LIN {X 0,Y 78.039,Z 374.236,A -85,B 0,C 180,E1 -30962.276,E2 -30962.276} C_VEL
LIN {X 0,Y 75.097,Z 386.191,A -85,B 0,C 180,E1 -30962.659,E2 -30962.659} C_VEL
LIN {X 0,Y 70.422,Z 399.419,A -85,B 0,C 180,E1 -30963.507,E2 -30963.507} C_VEL
LIN {X 0,Y 64.332,Z 411.877,A -85,B 0,C 180,E1 -30964.416,E2 -30964.416} C_VEL
LIN {X 0,Y 57.436,Z 423.118,A -85,B 0,C 180,E1 -30966.078,E2 -30966.078} C_VEL
LIN {X 0,Y 49.737,Z 433.18,A -85,B 0,C 180,E1 -30968.373,E2 -30968.373} C_VEL
LIN {X 0,Y 41.305,Z 442.293,A -85,B 0,C 180,E1 -30971.87,E2 -30971.87} C_VEL
LIN {X 0,Y 31.483,Z 451.164,A -85,B 0,C 180,E1 -30978.364,E2 -30978.364} C_VEL
LIN {X 0,Y 22.364,Z 458.209,A -85,B 0,C 180,E1 -30990.155,E2 -30990.155} C_VEL
LIN {X 0,Y 16.168,Z 463.002,A -85,B 0,C 180,E1 -31009.254,E2 -31009.254} C_VEL
LIN {X 0,Y 12.989,Z 467.557,A -85,B 0,C 180,E1 -31049.952,E2 -31049.952} C_VEL
LIN {X 0,Y 14.487,Z 469.9,A -85,B 0,C 180,E1 -31078.972,E2 -31078.972} C_VEL
LIN {X 0,Y 18.537,Z 471.807,A -85,B 0,C 180,E1 -31099.259,E2 -31099.259} C_VEL
LIN {X 0,Y 30.055,Z 474.427,A -85,B 0,C 180,E1 -31119.226,E2 -31119.226} C_VEL
LIN {X 0,Y 43.189,Z 475.464,A -85,B 0,C 180,E1 -31127.447,E2 -31127.447} C_VEL
LIN {X 0,Y 49.96,Z 475.43,A -85,B 0,C 180,E1 -31129.894,E2 -31129.894} C_VEL
LIN {X 0,Y 49.912,Z 475.428,A -85,B 0,C 180,E1 -31130.205,E2 -31130.205} C_VEL
LIN {X 0,Y 42.475,Z 475.388,A -85,B 0,C 180,E1 -31132.983,E2 -31132.983} C_VEL
LIN {X 0,Y 30.984,Z 474.383,A -85,B 0,C 180,E1 -31139.95,E2 -31139.95} C_VEL
LIN {X 0,Y 21.533,Z 472.495,A -85,B 0,C 180,E1 -31151.868,E2 -31151.868} C_VEL
LIN {X 0,Y 13.826,Z 469.451,A -85,B 0,C 180,E1 -31180.388,E2 -31180.388} C_VEL
LIN {X 0,Y 13.127,Z 465.27,A -85,B 0,C 180,E1 -31230.048,E2 -31230.048} C_VEL
LIN {X 0,Y 19.696,Z 459.87,A -85,B 0,C 180,E1 -31262.397,E2 -31262.397} C_VEL
LIN {X 0,Y 28.677,Z 453.089,A -85,B 0,C 180,E1 -31277.359,E2 -31277.359} C_VEL
LIN {X 0,Y 38.527,Z 444.654,A -85,B 0,C 180,E1 -31285.201,E2 -31285.201} C_VEL
LIN {X 0,Y 45.556,Z 437.596,A -85,B 0,C 180,E1 -31288.628,E2 -31288.628} C_VEL
LIN {X 0,Y 49.181,Z 433.304,A -85,B 0,C 180,E1 -31290.888,E2 -31290.888} C_VEL
LIN {X 0,Y 54.376,Z 425.964,A -85,B 0,C 180,E1 -31295.555,E2 -31295.555} C_VEL
LIN {X 0,Y 59.23,Z 418.141,A -85,B 0,C 180,E1 -31299.3,E2 -31299.3} C_VEL
LIN {X 0,Y 62.124,Z 413.092,A -85,B 0,C 180,E1 -31300.314,E2 -31300.314} C_VEL
LIN {X 0,Y 68.321,Z 400.856,A -85,B 0,C 180,E1 -31301.02,E2 -31301.02} C_VEL
LIN {X 0,Y 73.111,Z 388.298,A -85,B 0,C 180,E1 -31301.539,E2 -31301.539} C_VEL
LIN {X 0,Y 76.561,Z 375.283,A -85,B 0,C 180,E1 -31301.809,E2 -31301.809} C_VEL
LIN {X 0,Y 78.852,Z 360.598,A -85,B 0,C 180,E1 -31302.057,E2 -31302.057} C_VEL
LIN {X 0,Y 78.902,Z 359.79,A -85,B 0,C 180,E1 -31302.391,E2 -31302.391} C_VEL
LIN {X 0,Y 78.681,Z 357.8,A -85,B 0,C 180,E1 -31306.83,E2 -31306.83} C_VEL
LIN {X 0,Y 78.732,Z 357.243,A -85,B 0,C 180,E1 -31311.676,E2 -31311.676} C_VEL
LIN {X 0,Y 78.797,Z 357.715,A -85,B 0,C 180,E1 -31313.505,E2 -31313.505} C_VEL
LIN {X 0,Y 78.961,Z 359.812,A -85,B 0,C 180,E1 -31316.818,E2 -31316.818} C_VEL
LIN {X 0,Y 76.701,Z 374.738,A -85,B 0,C 180,E1 -31317.1,E2 -31317.1} C_VEL
LIN {X 0,Y 73.62,Z 386.882,A -85,B 0,C 180,E1 -31317.323,E2 -31317.323} C_VEL
LIN {X 0,Y 69.024,Z 399.468,A -85,B 0,C 180,E1 -31317.79,E2 -31317.79} C_VEL
LIN {X 0,Y 63.296,Z 411.104,A -85,B 0,C 180,E1 -31318.133,E2 -31318.133} C_VEL
LIN {X 0,Y 56.243,Z 422.472,A -85,B 0,C 180,E1 -31319.025,E2 -31319.025} C_VEL
LIN {X 0,Y 49.207,Z 431.659,A -85,B 0,C 180,E1 -31320.181,E2 -31320.181} C_VEL
LIN {X 0,Y 42.193,Z 439.291,A -85,B 0,C 180,E1 -31321.513,E2 -31321.513} C_VEL
LIN {X 0,Y 33.476,Z 447.315,A -85,B 0,C 180,E1 -31324.023,E2 -31324.023} C_VEL
LIN {X 0,Y 23.14,Z 455.107,A -85,B 0,C 180,E1 -31329.048,E2 -31329.048} C_VEL
LIN {X 0,Y 14.842,Z 460.427,A -85,B 0,C 180,E1 -31338.599,E2 -31338.599} C_VEL
LIN {X 0,Y 6.702,Z 465.536,A -85,B 0,C 180,E1 -31378.27,E2 -31378.27} C_VEL
LIN {X 0,Y 6.813,Z 468.237,A -85,B 0,C 180,E1 -31440.94,E2 -31440.94} C_VEL
LIN {X 0,Y 14.906,Z 471.387,A -85,B 0,C 180,E1 -31480.432,E2 -31480.432} C_VEL
LIN {X 0,Y 21.507,Z 472.952,A -85,B 0,C 180,E1 -31488.469,E2 -31488.469} C_VEL
LIN {X 0,Y 21.334,Z 472.903,A -85,B 0,C 180,E1 -31491.031,E2 -31491.031} C_VEL
LIN {X 0,Y 10.388,Z 469.916,A -85,B 0,C 180,E1 -31507.776,E2 -31507.776} C_VEL
LIN {X 0,Y 5.57,Z 465.952,A -85,B 0,C 180,E1 -31590.113,E2 -31590.113} C_VEL
LIN {X 0,Y 14,Z 460.712,A -85,B 0,C 180,E1 -31638.919,E2 -31638.919} C_VEL
LIN {X 0,Y 22.572,Z 455.326,A -85,B 0,C 180,E1 -31648.948,E2 -31648.948} C_VEL
LIN {X 0,Y 33.309,Z 447.267,A -85,B 0,C 180,E1 -31654.654,E2 -31654.654} C_VEL
LIN {X 0,Y 42.002,Z 439.322,A -85,B 0,C 180,E1 -31657.006,E2 -31657.006} C_VEL
LIN {X 0,Y 50.898,Z 429.391,A -85,B 0,C 180,E1 -31658.788,E2 -31658.788} C_VEL
LIN {X 0,Y 58.936,Z 418.316,A -85,B 0,C 180,E1 -31659.927,E2 -31659.927} C_VEL
LIN {X 0,Y 62.124,Z 413.092,A -85,B 0,C 180,E1 -31660.314,E2 -31660.314} C_VEL
LIN {X 0,Y 64.839,Z 407.98,A -85,B 0,C 180,E1 -31661.208,E2 -31661.208} C_VEL
LIN {X 0,Y 69.959,Z 395.85,A -85,B 0,C 180,E1 -31665.051,E2 -31665.051} C_VEL
LIN {X 0,Y 72.441,Z 388.634,A -85,B 0,C 180,E1 -31666.763,E2 -31666.763} C_VEL
LIN {X 0,Y 73.577,Z 384.881,A -85,B 0,C 180,E1 -31667.095,E2 -31667.095} C_VEL
LIN {X 0,Y 76.708,Z 371.669,A -85,B 0,C 180,E1 -31667.141,E2 -31667.141} C_VEL
LIN {X 0,Y 77.751,Z 364.818,A -85,B 0,C 180,E1 -31667.3,E2 -31667.3} C_VEL
LIN {X 0,Y 77.822,Z 364.302,A -85,B 0,C 180,E1 -31671.703,E2 -31671.703} C_VEL
LIN {X 0,Y 76.13,Z 374.628,A -85,B 0,C 180,E1 -31671.809,E2 -31671.809} C_VEL
LIN {X 0,Y 73.015,Z 386.845,A -85,B 0,C 180,E1 -31671.801,E2 -31671.801} C_VEL
LIN {X 0,Y 68.334,Z 399.525,A -85,B 0,C 180,E1 -31671.916,E2 -31671.916} C_VEL
LIN {X 0,Y 62.157,Z 411.918,A -85,B 0,C 180,E1 -31671.696,E2 -31671.696} C_VEL
LIN {X 0,Y 55.043,Z 423.101,A -85,B 0,C 180,E1 -31671.78,E2 -31671.78} C_VEL
LIN {X 0,Y 47.459,Z 432.674,A -85,B 0,C 180,E1 -31671.838,E2 -31671.838} C_VEL
LIN {X 0,Y 39.064,Z 441.392,A -85,B 0,C 180,E1 -31671.8,E2 -31671.8} C_VEL
LIN {X 0,Y 28.425,Z 450.386,A -85,B 0,C 180,E1 -31671.637,E2 -31671.637} C_VEL
LIN {X 0,Y 17.806,Z 457.574,A -85,B 0,C 180,E1 -31670.868,E2 -31670.868} C_VEL
LIN {X 0,Y 14.266,Z 459.617,A -85,B 0,C 180,E1 -31670.421,E2 -31670.421} C_VEL
LIN {X 0,Y 14.357,Z 459.56,A -85,B 0,C 180,E1 -31668.469,E2 -31668.469} C_VEL
LIN {X 0,Y 25.258,Z 452.665,A -85,B 0,C 180,E1 -31666.984,E2 -31666.984} C_VEL
LIN {X 0,Y 36.107,Z 444.099,A -85,B 0,C 180,E1 -31666.783,E2 -31666.783} C_VEL
LIN {X 0,Y 46.034,Z 434.228,A -85,B 0,C 180,E1 -31666.777,E2 -31666.777} C_VEL
LIN {X 0,Y 54.15,Z 424.268,A -85,B 0,C 180,E1 -31666.807,E2 -31666.807} C_VEL
LIN {X 0,Y 61.701,Z 412.713,A -85,B 0,C 180,E1 -31666.859,E2 -31666.859} C_VEL
LIN {X 0,Y 67.277,Z 401.854,A -85,B 0,C 180,E1 -31666.97,E2 -31666.97} C_VEL
LIN {X 0,Y 72.113,Z 389.554,A -85,B 0,C 180,E1 -31667.091,E2 -31667.091} C_VEL
LIN {X 0,Y 73.577,Z 384.881,A -85,B 0,C 180,E1 -31667.095,E2 -31667.095} C_VEL
LIN {X 0,Y 77.48,Z 385.443,A -85,B 0,C 180,E1 -31667.368,E2 -31667.368} C_VEL
LIN {X 0,Y 77.48,Z 600,A -85,B 0,C 180,E1 -31667.368,E2 -31667.368} C_VEL
LIN {X 0,Y 77.48,Z 600,A -85,B 0,C 180,E1 -31667.368,E2 -31667.368}

QRS_NEXT_CUT()

QRS_NEXT()
QRS_HOME()

END
